Universal Robots PolyScope program: ATI Demo Program.urp

Program ATI Demo Program (installation=default directory=/programs/usbdisk/20220721 createdIn=3.1.18024.0 lastSavedIn=3.15.6.106324 robotSerialNumber=2016353406)
Calibrated DH parameters: a=[0.000241, -0.156882, -0.391168, -0.000034, 0.000033, 0]; d=[0.08909, 1210.353649, -1202.089359, -8.154207, 0.094912, 0.082482]; alpha=[1.570962, 0.000326, -0.003342, 1.570446, -1.570439, 0]; deltaTheta=[0.000082, 1.192638, -1.263181, 0.0705, 0.00007, 0.000052]
BeforeStart
  Folder Move to Initial start position
    MoveJ speed 60 deg/s, acceleration 80 deg/s^2 (useActiveTCP=false)
      'CAUTION: check reachability or edit Waypoint before running Demo!'
      Waypoint Start: TCP in base x=-436.352 y=579.706 z=355.306 mm, rx=3.1399 ry=-0.0472 rz=-0.0056 rad; joints [-61.803, -57.175, 58.456, -91.289, 270.047, 29.954] deg
  URCap F/T Sensor Command (ATI Axia Force/Torque Sensor, ATI Industrial Automation) dataModel(WEIGHT=0.025, running=Enable)
  'Initialize variable for use in Thread:'
  'In this example, we name the variable ATI_FT_data.'
  ATI_FT_rawdata := ati_ftsensor.get_raw_ft()
Robot Program (runOnlyOnce=false)
  Folder Bias the sensor
    Wait Sleep waitTime=0.5
    URCap F/T Sensor Command (ATI Axia Force/Torque Sensor, ATI Industrial Automation) dataModel(running=Bias)
    Wait Sleep waitTime=0.5
  'This Demo program shows multiple ways to search & monitor forces (without UR Force Mode)'
  'and program offset motion with UR Force Mode.'
  Folder METHOD 1
    Folder Move down until the tool touches a surface
      'Monitor Norm of Forces (in robot base coordinate frame)'
      MoveL speed 40 mm/s, acceleration 200 mm/s^2 (useActiveTCP=false) feature=Base
        If ForceNorm<2 (checkContinuously=true)
          Waypoint RelativeMotionZ (Relative): relativeFromPosition TCP in base x=-99.537 y=-399.332 z=353.883 mm, rx=0.0027 ry=-3.1384 rz=-0.0008 rad; joints [-88.578, -78.615, -111.599, -79.821, 89.816, 1.322] deg; TCP in base x=-100.895 y=-399.448 z=-109.905 mm, rx=-0.0035 ry=-3.1383 rz=-0.0004 rad; joints [-88.578, -139.653, -133.528, 3.146, 89.816, 1.322] deg
    Folder Move across the surface while applying 10N of force
      'Use "Simple" type UR Force Control'
      Force Simple feature=Joint_6_name; selection=[0, 0, 1, 0, 0, 0]; wrench=[0, 0, 10, 0, 0, 0]; limitsForce=[0.15, 0.15, 0.15, 1.047198, 1.047198, 1.047198]; limitsMotion=[0.1, 0.1, 0.1, 0.349066, 0.349066, 0.349066]
        MoveL speed 40 mm/s, acceleration 25 mm/s^2 (useActiveTCP=false) feature=Joint_6_name
          Wait Sleep waitTime=1
          Folder (Optional IF) Stop if the tool encounters too much resistance or hits wall.
            If xyPlaneForce < 10 (checkContinuously=true)
              Waypoint RelativeMotionY (Relative): relativeFromPosition TCP in base x=-436.359 y=579.696 z=355.25 mm, rx=3.1399 ry=-0.0472 rz=-0.0054 rad; joints [-61.803, -57.175, 58.456, -91.289, 270.047, 29.954] deg; TCP in base x=436.38 y=579.622 z=355.372 mm, rx=3.1399 ry=-0.0472 rz=-0.0051 rad; joints [-135.73, -57.119, 58.32, -90.983, 269.918, -43.973] deg; flange x=436.37 y=579.672 z=355.256 mm, rx=3.1399 ry=-0.0472 rz=-0.0054 rad
      Folder Reset to a start position
        MoveL speed 250 mm/s, acceleration 1200 mm/s^2 (useActiveTCP=false) feature=Base
          Waypoint Up (Relative): relativeFromPosition TCP in base x=-436.39 y=579.651 z=262.908 mm, rx=3.1399 ry=-0.047 rz=-0.0055 rad; joints [-61.794, -55.361, 69.182, -103.829, 270.049, 29.921] deg; TCP in base x=-436.336 y=579.673 z=343.365 mm, rx=3.14 ry=-0.0472 rz=-0.0056 rad; joints [-61.802, -57.106, 60.102, -93.003, 270.047, 29.949] deg; flange x=-436.348 y=579.679 z=343.315 mm, rx=3.1399 ry=-0.0472 rz=-0.0055 rad
          SuppressedNode
            Waypoint firstUp: TCP in base x=436.386 y=579.646 z=286.859 mm, rx=3.1399 ry=-0.0472 rz=-0.0054 rad; joints [-135.724, -56.056, 66.674, -100.399, 269.918, -43.997] deg
          Waypoint Start: TCP in base x=-436.352 y=579.706 z=355.306 mm, rx=3.1399 ry=-0.0472 rz=-0.0056 rad; joints [-61.803, -57.175, 58.456, -91.289, 270.047, 29.954] deg
  Folder Reset to a start position
    MoveL speed 250 mm/s, acceleration 1200 mm/s^2 (useActiveTCP=false) feature=Base
      Waypoint Start: TCP in base x=-436.352 y=579.706 z=355.306 mm, rx=3.1399 ry=-0.0472 rz=-0.0056 rad; joints [-61.803, -57.175, 58.456, -91.289, 270.047, 29.954] deg
  Folder METHOD 2
    Folder Move down until the tool touches a surface
      'Monitor Norm of Forces (in robot base coordinate frame)'
      MoveL speed 40 mm/s, acceleration 200 mm/s^2 (useActiveTCP=false) feature=Base
        If ForceNorm<2 (checkContinuously=true)
          Waypoint RelativeMotionZ (Relative): relativeFromPosition TCP in base x=-99.537 y=-399.332 z=353.883 mm, rx=0.0027 ry=-3.1384 rz=-0.0008 rad; joints [-88.578, -78.615, -111.599, -79.821, 89.816, 1.322] deg; TCP in base x=-100.895 y=-399.448 z=-109.905 mm, rx=-0.0035 ry=-3.1383 rz=-0.0004 rad; joints [-88.578, -139.653, -133.528, 3.146, 89.816, 1.322] deg
    Folder Move across the surface while applying 10N of down force & 0N of side force
      'Use "Motion" type UR Force Control with only Z compliance'
      Force Motion feature=Joint_6_name; selection=[0, 0, 1, 0, 0, 0]; wrench=[0, 0, 10, 0, 0, 0]; limitsForce=[0.15, 0.15, 0.15, 1.047198, 1.047198, 1.047198]; limitsMotion=[0.1, 0.1, 0.1, 0.349066, 0.349066, 0.349066]
        MoveL speed 40 mm/s, acceleration 25 mm/s^2 (useActiveTCP=true) feature=Base
          Wait Sleep waitTime=1
          Folder (Optional IF) Stop if the tool encounters too much resistance or hits wall.
            If xyPlaneForce < 10 (checkContinuously=true)
              Waypoint RelativeMotionY (Relative): relativeFromPosition TCP in base x=-436.359 y=579.696 z=355.25 mm, rx=3.1399 ry=-0.0472 rz=-0.0054 rad; joints [-61.803, -57.175, 58.456, -91.289, 270.047, 29.954] deg; TCP in base x=436.38 y=579.622 z=355.372 mm, rx=3.1399 ry=-0.0472 rz=-0.0051 rad; joints [-135.73, -57.119, 58.32, -90.983, 269.918, -43.973] deg; flange x=436.37 y=579.672 z=355.256 mm, rx=3.1399 ry=-0.0472 rz=-0.0054 rad
      Folder Reset to a start position
        MoveL speed 250 mm/s, acceleration 1200 mm/s^2 (useActiveTCP=false) feature=Base
          Waypoint Up (Relative): relativeFromPosition TCP in base x=-436.39 y=579.651 z=262.908 mm, rx=3.1399 ry=-0.047 rz=-0.0055 rad; joints [-61.794, -55.361, 69.182, -103.829, 270.049, 29.921] deg; TCP in base x=-436.336 y=579.673 z=343.365 mm, rx=3.14 ry=-0.0472 rz=-0.0056 rad; joints [-61.802, -57.106, 60.102, -93.003, 270.047, 29.949] deg; flange x=-436.348 y=579.679 z=343.315 mm, rx=3.1399 ry=-0.0472 rz=-0.0055 rad
          SuppressedNode
            Waypoint firstUp: TCP in base x=436.386 y=579.646 z=286.859 mm, rx=3.1399 ry=-0.0472 rz=-0.0054 rad; joints [-135.724, -56.056, 66.674, -100.399, 269.918, -43.997] deg
          Waypoint Start: TCP in base x=-436.352 y=579.706 z=355.306 mm, rx=3.1399 ry=-0.0472 rz=-0.0056 rad; joints [-61.803, -57.175, 58.456, -91.289, 270.047, 29.954] deg
  Folder Reset to a start position
    MoveL speed 250 mm/s, acceleration 1200 mm/s^2 (useActiveTCP=false) feature=Base
      Waypoint Start: TCP in base x=-436.352 y=579.706 z=355.306 mm, rx=3.1399 ry=-0.0472 rz=-0.0056 rad; joints [-61.803, -57.175, 58.456, -91.289, 270.047, 29.954] deg
  Folder METHOD 3
    Folder Move down until the tool touches a surface
      'Monitor Norm of Forces (in robot base coordinate frame)'
      MoveL speed 40 mm/s, acceleration 200 mm/s^2 (useActiveTCP=false) feature=Base
        If ForceNorm<2 (checkContinuously=true)
          Waypoint RelativeMotionZ (Relative): relativeFromPosition TCP in base x=-99.537 y=-399.332 z=353.883 mm, rx=0.0027 ry=-3.1384 rz=-0.0008 rad; joints [-88.578, -78.615, -111.599, -79.821, 89.816, 1.322] deg; TCP in base x=-100.895 y=-399.448 z=-109.905 mm, rx=-0.0035 ry=-3.1383 rz=-0.0004 rad; joints [-88.578, -139.653, -133.528, 3.146, 89.816, 1.322] deg
    Folder Move across the surface while applying 10N of force
      'Use "Motion" type UR Force Control with Y & Z compliance, only push in Z'
      Force Motion feature=Joint_6_name; selection=[0, 1, 1, 0, 0, 0]; wrench=[0, 0, 10, 0, 0, 0]; limitsForce=[0.15, 0.15, 0.15, 1.047198, 1.047198, 1.047198]; limitsMotion=[0.1, 0.1, 0.1, 0.349066, 0.349066, 0.349066]
        MoveL speed 40 mm/s, acceleration 25 mm/s^2 (useActiveTCP=true) feature=Base
          Wait Sleep waitTime=1
          Folder (Optional IF) Stop if the tool encounters too much resistance or hits wall.
            If xyPlaneForce < 10 (checkContinuously=true)
              Waypoint RelativeMotionY (Relative): relativeFromPosition TCP in base x=-436.359 y=579.696 z=355.25 mm, rx=3.1399 ry=-0.0472 rz=-0.0054 rad; joints [-61.803, -57.175, 58.456, -91.289, 270.047, 29.954] deg; TCP in base x=436.38 y=579.622 z=355.372 mm, rx=3.1399 ry=-0.0472 rz=-0.0051 rad; joints [-135.73, -57.119, 58.32, -90.983, 269.918, -43.973] deg; flange x=436.37 y=579.672 z=355.256 mm, rx=3.1399 ry=-0.0472 rz=-0.0054 rad
      Folder Reset to a start position
        MoveL speed 250 mm/s, acceleration 1200 mm/s^2 (useActiveTCP=false) feature=Base
          Waypoint Up (Relative): relativeFromPosition TCP in base x=-436.39 y=579.651 z=262.908 mm, rx=3.1399 ry=-0.047 rz=-0.0055 rad; joints [-61.794, -55.361, 69.182, -103.829, 270.049, 29.921] deg; TCP in base x=-436.336 y=579.673 z=343.365 mm, rx=3.14 ry=-0.0472 rz=-0.0056 rad; joints [-61.802, -57.106, 60.102, -93.003, 270.047, 29.949] deg; flange x=-436.348 y=579.679 z=343.315 mm, rx=3.1399 ry=-0.0472 rz=-0.0055 rad
          SuppressedNode
            Waypoint firstUp: TCP in base x=436.386 y=579.646 z=286.859 mm, rx=3.1399 ry=-0.0472 rz=-0.0054 rad; joints [-135.724, -56.056, 66.674, -100.399, 269.918, -43.997] deg
          Waypoint Start: TCP in base x=-436.352 y=579.706 z=355.306 mm, rx=3.1399 ry=-0.0472 rz=-0.0056 rad; joints [-61.803, -57.175, 58.456, -91.289, 270.047, 29.954] deg
  Folder Reset to a start position
    MoveL speed 250 mm/s, acceleration 1200 mm/s^2 (useActiveTCP=false) feature=Base
      Waypoint Start: TCP in base x=-436.352 y=579.706 z=355.306 mm, rx=3.1399 ry=-0.0472 rz=-0.0056 rad; joints [-61.803, -57.175, 58.456, -91.289, 270.047, 29.954] deg
  Folder METHOD 4
    Folder Move down until the tool touches a surface
      'Monitor raw FT sensor readings (in sensor coordinate frame)'
      MoveL speed 40 mm/s, acceleration 200 mm/s^2 (useActiveTCP=false) feature=Base
        If ATI_FT_Fz>-2 (checkContinuously=true)
          Waypoint RelativeMotionZ (Relative): relativeFromPosition TCP in base x=-99.537 y=-399.332 z=353.883 mm, rx=0.0027 ry=-3.1384 rz=-0.0008 rad; joints [-88.578, -78.615, -111.599, -79.821, 89.816, 1.322] deg; TCP in base x=-100.895 y=-399.448 z=-109.905 mm, rx=-0.0035 ry=-3.1383 rz=-0.0004 rad; joints [-88.578, -139.653, -133.528, 3.146, 89.816, 1.322] deg
      Wait Sleep waitTime=2
    '(Optional) Insert a UR Force Mode command to move across the surface, as shown in Methods above.'
    Folder Reset to a start position
      MoveL speed 150 mm/s, acceleration 400 mm/s^2 (useActiveTCP=false) feature=Base
        Waypoint Up (Relative): relativeFromPosition TCP in base x=-436.39 y=579.651 z=262.908 mm, rx=3.1399 ry=-0.047 rz=-0.0055 rad; joints [-61.794, -55.361, 69.182, -103.829, 270.049, 29.921] deg; TCP in base x=-436.336 y=579.673 z=343.365 mm, rx=3.14 ry=-0.0472 rz=-0.0056 rad; joints [-61.802, -57.106, 60.102, -93.003, 270.047, 29.949] deg; flange x=-436.348 y=579.679 z=343.315 mm, rx=3.1399 ry=-0.0472 rz=-0.0055 rad
        SuppressedNode
          Waypoint secondUp: TCP in base x=-436.356 y=579.68 z=269.926 mm, rx=3.1399 ry=-0.047 rz=-0.0055 rad; joints [-61.795, -55.594, 68.513, -102.927, 270.049, 29.924] deg
        Waypoint Start: TCP in base x=-436.352 y=579.706 z=355.306 mm, rx=3.1399 ry=-0.0472 rz=-0.0056 rad; joints [-61.803, -57.175, 58.456, -91.289, 270.047, 29.954] deg
Thread Thread_1 (runOnlyOnce=false)
  'MONITOR THIS DATA DURING PROGRAM FROM "Variables" TAB'
  Wait Sleep waitTime=0.01
  'Read sensor F/T Data using F/T URCap command, & assign it to a variable.'
  'This is the raw data directly from the sensor, in the sensor coordinate frame.'
  'With every loop of the thread, update the raw F/T data reading.'
  ATI_FT_rawdata := ati_ftsensor.get_raw_ft()
  'Fz is the 3rd element of the ATI_FT_data variable.'
  'NOTE: Pressing sensor in Z causes a -Z force (if no sensor Tool Transform applied)'
  ATI_FT_Fz := ATI_FT_rawdata[2]
  'F/T sensor data can also be read from native UR commands.'
  'Data read from UR commands will have transformations applied.'
  '(it is in robot base frame, not in the sensor coordinate frame).'
  ' UR Command get_tcp_force() gives TCP force in coordinate frame of robot base.'
  FTinBaseFrame := get_tcp_force()
  'UR command force() gives the Norm of get_tcp_force().'
  ForceNorm := force()
  Folder Get magnitude of force in just the X-Y plane, accounting for friction of tool
    xyPlaneForce := sqrt(pow(FTinBaseFrame[0], 2) + pow(FTinBaseFrame[1], 2)) - 0.3*ForceNorm
